// TIA Portal V19 export
FUNCTION "FC_Hilfsfuntionen" : Void   // FC169, LAD
TITLE = Hilfsfunktionen
{ S7_Optimized_Access := 'TRUE' }
// stored: AutoNumber false, SetENOAutomatically true
   VAR_TEMP
      Anf_links : Bool;
      Anf_rechts : Bool;
      Niv_CM01_ok : Bool;
      Niv_CM02_ok : Bool;
      Niv_Spuelen_ok : Bool;
      Fuellstand_ok : Bool;
      Nr : Int;
   END_VAR
   VAR CONSTANT
      Typ_KSoLS : Byte := 16#10;
      Typ_KS : Byte := 16#11;
      Typ_LS : Byte := 16#12;
      Typ_GO_Sperre : Byte := 16#13;
      Typ_GO : Byte := 16#20;
      Ausfahrt : Byte := 16#19;
   END_VAR
BEGIN

REGION Network 1 (SCL): Einfahrsperren / Detailtypen
   REGION CM01
       // CM01 komplett leer
       IF NOT "DB_POS".POS[1].belegt AND NOT NOT "DB_POS".POS[2].belegt AND NOT "DB_POS".POS[3].belegt AND NOT "DB_POS".POS[4].belegt AND NOT "DB_POS".POS[5].belegt AND NOT "DB_POS".POS[6].belegt THEN
           "DB_POS".POS[1].notFG_in := FALSE;
           "DB_POS".POS[2].notFG_in := FALSE;
           "DB_POS".POS[5].notFG_in := FALSE;
           "DB_POS".POS[6].notFG_in := FALSE;
           "DB_POS".POS[1].Detailtyp := #Typ_KSoLS;
           "DB_POS".POS[2].Detailtyp := #Typ_KSoLS;
           "DB_POS".POS[5].Detailtyp := #Typ_KSoLS;
           "DB_POS".POS[6].Detailtyp := #Typ_KSoLS;
       END_IF;
       // Pos.3 (GO) Ziel bzw. belegt
       IF "DB_POS".POS[3].next_WT <> 0 THEN
           "DB_POS".POS[1].notFG_in := TRUE;
           "DB_POS".POS[5].notFG_in := TRUE;
           "DB_POS".POS[1].Detailtyp := #Typ_GO_Sperre;
           "DB_POS".POS[5].Detailtyp := #Typ_GO_Sperre;
       ELSE
           "DB_POS".POS[1].notFG_in := FALSE;
           "DB_POS".POS[5].notFG_in := FALSE;
           "DB_POS".POS[1].Detailtyp := #Typ_KSoLS;
           "DB_POS".POS[5].Detailtyp := #Typ_KSoLS;
       END_IF;
       // Pos.4 (GO) Ziel bzw. belegt 
       IF "DB_POS".POS[4].next_WT <> 0 THEN
           "DB_POS".POS[2].notFG_in := TRUE;
           "DB_POS".POS[6].notFG_in := TRUE;
           "DB_POS".POS[2].Detailtyp := #Typ_GO_Sperre;
           "DB_POS".POS[6].Detailtyp := #Typ_GO_Sperre;
       ELSE
           "DB_POS".POS[2].notFG_in := FALSE;
           "DB_POS".POS[6].notFG_in := FALSE;
           "DB_POS".POS[2].Detailtyp := #Typ_KSoLS;
           "DB_POS".POS[6].Detailtyp := #Typ_KSoLS;
       END_IF;
       //Pos.1/2
       IF ("DB_POS".POS[1].next_WT <> 0) AND ("DB_POS".POS[1].next_WT = "DB_POS".POS[2].next_WT) THEN
           "DB_POS".POS[1].Detailtyp := #Typ_LS;
           "DB_POS".POS[2].Detailtyp := #Typ_LS;
       ELSIF ("DB_POS".POS[1].next_WT <> 0) OR ("DB_POS".POS[2].next_WT <> 0) THEN
           "DB_POS".POS[1].Detailtyp := #Typ_KS;
           "DB_POS".POS[2].Detailtyp := #Typ_KS;
       END_IF;
       //Pos.5/6
       IF ("DB_POS".POS[5].next_WT <> 0) AND ("DB_POS".POS[5].next_WT = "DB_POS".POS[6].next_WT) THEN
           "DB_POS".POS[5].Detailtyp := #Typ_LS;
           "DB_POS".POS[6].Detailtyp := #Typ_LS;
       ELSIF ("DB_POS".POS[5].next_WT <> 0) OR ("DB_POS".POS[6].next_WT <> 0) THEN
           "DB_POS".POS[5].Detailtyp := #Typ_KS;
           "DB_POS".POS[6].Detailtyp := #Typ_KS;
       END_IF;
       //Einfahrsperre Pos.3/4
       "DB_POS".POS[3].notFG_in := ("DB_POS".POS[1].next_WT <> 0) OR ("DB_POS".POS[5].next_WT <> 0);
       "DB_POS".POS[4].notFG_in := ("DB_POS".POS[2].next_WT <> 0) OR ("DB_POS".POS[6].next_WT <> 0);
   END_REGION

   REGION CM03
       // CM03 komplett leer
       IF NOT "DB_POS".POS[7].belegt AND NOT NOT "DB_POS".POS[8].belegt AND NOT "DB_POS".POS[9].belegt AND NOT "DB_POS".POS[10].belegt AND NOT "DB_POS".POS[11].belegt AND NOT "DB_POS".POS[12].belegt THEN
           "DB_POS".POS[7].notFG_in := FALSE;
           "DB_POS".POS[8].notFG_in := FALSE;
           "DB_POS".POS[11].notFG_in := FALSE;
           "DB_POS".POS[12].notFG_in := FALSE;
           "DB_POS".POS[7].Detailtyp := #Typ_KSoLS;
           "DB_POS".POS[8].Detailtyp := #Typ_KSoLS;
           "DB_POS".POS[11].Detailtyp := #Typ_KSoLS;
           "DB_POS".POS[12].Detailtyp := #Typ_KSoLS;
       END_IF;
       // Pos.9 (GO) Ziel bzw. belegt
       IF "DB_POS".POS[9].next_WT <> 0 THEN
           "DB_POS".POS[7].notFG_in := TRUE;
           "DB_POS".POS[11].notFG_in := TRUE;
           "DB_POS".POS[7].Detailtyp := #Typ_GO_Sperre;
           "DB_POS".POS[11].Detailtyp := #Typ_GO_Sperre;
       ELSE
           "DB_POS".POS[7].notFG_in := FALSE;
           "DB_POS".POS[11].notFG_in := FALSE;
           "DB_POS".POS[7].Detailtyp := #Typ_KSoLS;
           "DB_POS".POS[11].Detailtyp := #Typ_KSoLS;
       END_IF;
       // Pos.10 (GO) Ziel bzw. belegt 
       IF "DB_POS".POS[10].next_WT <> 0 THEN
           "DB_POS".POS[8].notFG_in := TRUE;
           "DB_POS".POS[12].notFG_in := TRUE;
           "DB_POS".POS[8].Detailtyp := #Typ_GO_Sperre;
           "DB_POS".POS[12].Detailtyp := #Typ_GO_Sperre;
       ELSE
           "DB_POS".POS[8].notFG_in := FALSE;
           "DB_POS".POS[12].notFG_in := FALSE;
           "DB_POS".POS[8].Detailtyp := #Typ_KSoLS;
           "DB_POS".POS[12].Detailtyp := #Typ_KSoLS;
       END_IF;
       //Pos.7/8
       IF ("DB_POS".POS[7].next_WT <> 0) AND ("DB_POS".POS[7].next_WT = "DB_POS".POS[8].next_WT) THEN
           "DB_POS".POS[7].Detailtyp := #Typ_LS;
           "DB_POS".POS[8].Detailtyp := #Typ_LS;
       ELSIF ("DB_POS".POS[7].next_WT <> 0) OR ("DB_POS".POS[8].next_WT <> 0) THEN
           "DB_POS".POS[7].Detailtyp := #Typ_KS;
           "DB_POS".POS[8].Detailtyp := #Typ_KS;
       END_IF;
       //Pos.11/12
       IF ("DB_POS".POS[11].next_WT <> 0) AND ("DB_POS".POS[11].next_WT = "DB_POS".POS[12].next_WT) THEN
           "DB_POS".POS[11].Detailtyp := #Typ_LS;
           "DB_POS".POS[12].Detailtyp := #Typ_LS;
       ELSIF ("DB_POS".POS[11].next_WT <> 0) OR ("DB_POS".POS[12].next_WT <> 0) THEN
           "DB_POS".POS[11].Detailtyp := #Typ_KS;
           "DB_POS".POS[12].Detailtyp := #Typ_KS;
       END_IF;
       //Einfahrsperre Pos.9/10
       "DB_POS".POS[9].notFG_in := ("DB_POS".POS[7].next_WT <> 0) OR ("DB_POS".POS[11].next_WT <> 0);
       "DB_POS".POS[10].notFG_in := ("DB_POS".POS[8].next_WT <> 0) OR ("DB_POS".POS[12].next_WT <> 0);
   END_REGION

   REGION CM02
       // CM02 komplett leer
       IF NOT "DB_POS".POS[13].belegt AND NOT NOT "DB_POS".POS[14].belegt AND NOT "DB_POS".POS[15].belegt AND NOT "DB_POS".POS[16].belegt AND NOT "DB_POS".POS[17].belegt AND NOT "DB_POS".POS[18].belegt THEN
           "DB_POS".POS[13].notFG_in := FALSE;
           "DB_POS".POS[14].notFG_in := FALSE;
           "DB_POS".POS[17].notFG_in := FALSE;
           "DB_POS".POS[18].notFG_in := FALSE;
           "DB_POS".POS[13].Detailtyp := #Typ_KSoLS;
           "DB_POS".POS[14].Detailtyp := #Typ_KSoLS;
           "DB_POS".POS[17].Detailtyp := #Typ_KSoLS;
           "DB_POS".POS[18].Detailtyp := #Typ_KSoLS;
       END_IF;
       // Pos.15 (GO) Ziel bzw. belegt
       IF "DB_POS".POS[15].next_WT <> 0 THEN
           "DB_POS".POS[13].notFG_in := TRUE;
           "DB_POS".POS[17].notFG_in := TRUE;
           "DB_POS".POS[13].Detailtyp := #Typ_GO_Sperre;
           "DB_POS".POS[17].Detailtyp := #Typ_GO_Sperre;
       ELSE
           "DB_POS".POS[13].notFG_in := FALSE;
           "DB_POS".POS[17].notFG_in := FALSE;
           "DB_POS".POS[13].Detailtyp := #Typ_KSoLS;
           "DB_POS".POS[17].Detailtyp := #Typ_KSoLS;
       END_IF;
       // Pos.16 (GO) Ziel bzw. belegt 
       IF "DB_POS".POS[16].next_WT <> 0 THEN
           "DB_POS".POS[14].notFG_in := TRUE;
           "DB_POS".POS[18].notFG_in := TRUE;
           "DB_POS".POS[14].Detailtyp := #Typ_GO_Sperre;
           "DB_POS".POS[18].Detailtyp := #Typ_GO_Sperre;
       ELSE
           "DB_POS".POS[14].notFG_in := FALSE;
           "DB_POS".POS[18].notFG_in := FALSE;
           "DB_POS".POS[14].Detailtyp := #Typ_KSoLS;
           "DB_POS".POS[18].Detailtyp := #Typ_KSoLS;
       END_IF;
       //Pos.13/14
       IF ("DB_POS".POS[13].next_WT <> 0) AND ("DB_POS".POS[13].next_WT = "DB_POS".POS[14].next_WT) THEN
           "DB_POS".POS[13].Detailtyp := #Typ_LS;
           "DB_POS".POS[14].Detailtyp := #Typ_LS;
       ELSIF ("DB_POS".POS[13].next_WT <> 0) OR ("DB_POS".POS[14].next_WT <> 0) THEN
           "DB_POS".POS[13].Detailtyp := #Typ_KS;
           "DB_POS".POS[14].Detailtyp := #Typ_KS;
       END_IF;
       //Pos.17/18
       IF ("DB_POS".POS[17].next_WT <> 0) AND ("DB_POS".POS[17].next_WT = "DB_POS".POS[18].next_WT) THEN
           "DB_POS".POS[17].Detailtyp := #Typ_LS;
           "DB_POS".POS[18].Detailtyp := #Typ_LS;
       ELSIF ("DB_POS".POS[17].next_WT <> 0) OR ("DB_POS".POS[18].next_WT <> 0) THEN
           "DB_POS".POS[17].Detailtyp := #Typ_KS;
           "DB_POS".POS[18].Detailtyp := #Typ_KS;
       END_IF;
       //Einfahrsperre Pos.15/16
       "DB_POS".POS[15].notFG_in := ("DB_POS".POS[13].next_WT <> 0) OR ("DB_POS".POS[17].next_WT <> 0);
       "DB_POS".POS[16].notFG_in := ("DB_POS".POS[14].next_WT <> 0) OR ("DB_POS".POS[18].next_WT <> 0);
   END_REGION

   REGION CM04
       // CM04 komplett leer
       IF NOT "DB_POS".POS[19].belegt AND NOT NOT "DB_POS".POS[20].belegt AND NOT "DB_POS".POS[21].belegt AND NOT "DB_POS".POS[22].belegt AND NOT "DB_POS".POS[23].belegt AND NOT "DB_POS".POS[24].belegt THEN
           "DB_POS".POS[19].notFG_in := FALSE;
           "DB_POS".POS[20].notFG_in := FALSE;
           "DB_POS".POS[23].notFG_in := FALSE;
           "DB_POS".POS[24].notFG_in := FALSE;
           "DB_POS".POS[19].Detailtyp := #Typ_KSoLS;
           "DB_POS".POS[20].Detailtyp := #Typ_KSoLS;
           "DB_POS".POS[23].Detailtyp := #Typ_KSoLS;
           "DB_POS".POS[24].Detailtyp := #Typ_KSoLS;
       END_IF;
       // Pos.21 (GO) Ziel bzw. belegt
       IF "DB_POS".POS[21].next_WT <> 0 THEN
           "DB_POS".POS[19].notFG_in := TRUE;
           "DB_POS".POS[23].notFG_in := TRUE;
           "DB_POS".POS[19].Detailtyp := #Typ_GO_Sperre;
           "DB_POS".POS[23].Detailtyp := #Typ_GO_Sperre;
       ELSE
           "DB_POS".POS[19].notFG_in := FALSE;
           "DB_POS".POS[23].notFG_in := FALSE;
           "DB_POS".POS[19].Detailtyp := #Typ_KSoLS;
           "DB_POS".POS[23].Detailtyp := #Typ_KSoLS;
       END_IF;
       // Pos.22 (GO) Ziel bzw. belegt 
       IF "DB_POS".POS[22].next_WT <> 0 THEN
           "DB_POS".POS[20].notFG_in := TRUE;
           "DB_POS".POS[24].notFG_in := TRUE;
           "DB_POS".POS[20].Detailtyp := #Typ_GO_Sperre;
           "DB_POS".POS[24].Detailtyp := #Typ_GO_Sperre;
       ELSE
           "DB_POS".POS[20].notFG_in := FALSE;
           "DB_POS".POS[24].notFG_in := FALSE;
           "DB_POS".POS[20].Detailtyp := #Typ_KSoLS;
           "DB_POS".POS[24].Detailtyp := #Typ_KSoLS;
       END_IF;
       //Pos.19/20
       IF ("DB_POS".POS[19].next_WT <> 0) AND ("DB_POS".POS[19].next_WT = "DB_POS".POS[20].next_WT) THEN
           "DB_POS".POS[19].Detailtyp := #Typ_LS;
           "DB_POS".POS[20].Detailtyp := #Typ_LS;
       ELSIF ("DB_POS".POS[19].next_WT <> 0) OR ("DB_POS".POS[20].next_WT <> 0) THEN
           "DB_POS".POS[19].Detailtyp := #Typ_KS;
           "DB_POS".POS[20].Detailtyp := #Typ_KS;
       END_IF;
       //Pos.23/24
       IF ("DB_POS".POS[23].next_WT <> 0) AND ("DB_POS".POS[23].next_WT = "DB_POS".POS[24].next_WT) THEN
           "DB_POS".POS[23].Detailtyp := #Typ_LS;
           "DB_POS".POS[24].Detailtyp := #Typ_LS;
       ELSIF ("DB_POS".POS[23].next_WT <> 0) OR ("DB_POS".POS[24].next_WT <> 0) THEN
           "DB_POS".POS[23].Detailtyp := #Typ_KS;
           "DB_POS".POS[24].Detailtyp := #Typ_KS;
       END_IF;
       //Einfahrsperre Pos.21/22
       "DB_POS".POS[21].notFG_in := ("DB_POS".POS[19].next_WT <> 0) OR ("DB_POS".POS[23].next_WT <> 0);
       "DB_POS".POS[22].notFG_in := ("DB_POS".POS[20].next_WT <> 0) OR ("DB_POS".POS[24].next_WT <> 0);
   END_REGION

   REGION Übergabe
       // Übergabe komplett leer
       IF NOT "DB_POS".POS[25].belegt AND NOT NOT "DB_POS".POS[26].belegt AND NOT "DB_POS".POS[27].belegt AND NOT "DB_POS".POS[28].belegt AND NOT "DB_POS".POS[29].belegt AND NOT "DB_POS".POS[30].belegt THEN
           "DB_POS".POS[25].Detailtyp := #Typ_KSoLS;
           "DB_POS".POS[26].Detailtyp := #Typ_KSoLS;
           "DB_POS".POS[29].Detailtyp := #Typ_KSoLS;
           "DB_POS".POS[30].Detailtyp := #Typ_KSoLS;
       END_IF;
       // Pos.27 (GO) Ziel bzw. belegt
       IF "DB_POS".POS[27].next_WT <> 0 THEN
           "DB_POS".POS[25].Detailtyp := #Typ_GO_Sperre;
           "DB_POS".POS[29].Detailtyp := #Typ_GO_Sperre;
       ELSE
           "DB_POS".POS[25].Detailtyp := #Typ_KSoLS;
           "DB_POS".POS[29].Detailtyp := #Typ_KSoLS;
       END_IF;
       // Pos.22 (GO) Ziel bzw. belegt 
       IF "DB_POS".POS[28].next_WT <> 0 THEN
           "DB_POS".POS[26].Detailtyp := #Typ_GO_Sperre;
           "DB_POS".POS[30].Detailtyp := #Typ_GO_Sperre;
       ELSE
           "DB_POS".POS[26].Detailtyp := #Typ_KSoLS;
           "DB_POS".POS[30].Detailtyp := #Typ_KSoLS;
       END_IF;
       //Pos.25/26
       IF ("DB_POS".POS[25].next_WT <> 0) AND ("DB_POS".POS[25].next_WT = "DB_POS".POS[26].next_WT) THEN
           "DB_POS".POS[25].Detailtyp := #Typ_LS;
           "DB_POS".POS[26].Detailtyp := #Typ_LS;
       ELSIF ("DB_POS".POS[25].next_WT <> 0) OR ("DB_POS".POS[26].next_WT <> 0) THEN
           "DB_POS".POS[25].Detailtyp := #Typ_KS;
           "DB_POS".POS[26].Detailtyp := #Typ_KS;
       END_IF;
       //Pos.29/30
       IF ("DB_POS".POS[29].next_WT <> 0) AND ("DB_POS".POS[29].next_WT = "DB_POS".POS[30].next_WT) THEN
           "DB_POS".POS[29].Detailtyp := #Typ_LS;
           "DB_POS".POS[30].Detailtyp := #Typ_LS;
       ELSIF ("DB_POS".POS[29].next_WT <> 0) OR ("DB_POS".POS[30].next_WT <> 0) THEN
           "DB_POS".POS[29].Detailtyp := #Typ_KS;
           "DB_POS".POS[30].Detailtyp := #Typ_KS;
       END_IF;

   END_REGION
END_REGION

REGION Network 2 (SCL): Deckelanforderungen

   REGION CM01
       #Anf_links := FALSE;
       #Anf_rechts := FALSE;

       // Check Quelle
       IF ("DB_POS".POS[1].Quelle AND ("DB_POS".POS[1].WT_DB <> 0)) OR
          ("DB_POS".POS[3].Quelle AND ("DB_POS".POS[3].WT_DB <> 0)) OR
          ("DB_POS".POS[5].Quelle AND  ("DB_POS".POS[5].WT_DB <> 0)) THEN
           #Anf_links := TRUE;
       END_IF;

       IF ("DB_POS".POS[2].Quelle AND ("DB_POS".POS[2].WT_DB <> 0)) OR
           ("DB_POS".POS[4].Quelle AND ("DB_POS".POS[4].WT_DB <> 0)) OR
           ("DB_POS".POS[6].Quelle AND  ("DB_POS".POS[6].WT_DB <> 0)) THEN
           #Anf_rechts := TRUE;
       END_IF;

       IF "DB_POS".POS[1].Quelle AND ("DB_POS".POS[1].WT_DB <> 0) AND ("DB_POS".POS[1].WT_DB = "DB_POS".POS[2].WT_DB) THEN
           #Anf_rechts := TRUE;
       END_IF;

       IF "DB_POS".POS[5].Quelle AND ("DB_POS".POS[5].WT_DB <> 0) AND ("DB_POS".POS[5].WT_DB = "DB_POS".POS[6].WT_DB) THEN
           #Anf_rechts := TRUE;
       END_IF;

       // Check Ziel
       IF (("DB_POS".POS[1].Ziel AND ("DB_POS".POS[1].next_WT <> 0)) OR ("DB_POS".POS[3].Ziel AND ("DB_POS".POS[3].next_WT <> 0)) OR ("DB_POS".POS[5].Ziel AND  ("DB_POS".POS[5].next_WT <> 0))) AND "DI_FW_1".ZST.Oben_li THEN
           #Anf_links := TRUE;
       END_IF;

       IF (("DB_POS".POS[2].Ziel AND ("DB_POS".POS[2].next_WT <> 0)) OR ("DB_POS".POS[4].Ziel AND ("DB_POS".POS[4].next_WT <> 0)) OR ("DB_POS".POS[6].Ziel AND  ("DB_POS".POS[6].next_WT <> 0)))  AND "DI_FW_1".ZST.Oben_re THEN
           #Anf_rechts := TRUE;
       END_IF;

       IF "DB_POS".POS[1].Ziel AND ("DB_POS".POS[1].next_WT <> 0) AND ("DB_POS".POS[1].next_WT = "DB_POS".POS[2].next_WT)  AND "DI_FW_1".ZST.Oben_re THEN
           #Anf_rechts := TRUE;
       END_IF;

       IF "DB_POS".POS[5].Ziel AND ("DB_POS".POS[5].next_WT <> 0) AND ("DB_POS".POS[5].next_WT = "DB_POS".POS[6].next_WT)  AND "DI_FW_1".ZST.Oben_re THEN
           #Anf_rechts := TRUE;
       END_IF;
       //
       IF #Anf_links THEN
           "Deckel_CM01".Zst.Req_links_auf := TRUE;
       ELSIF "Deckel_CM01".Zst.TW_sicher THEN
           "Deckel_CM01".Zst.Req_links_auf := FALSE;
       END_IF;

       IF #Anf_rechts THEN
           "Deckel_CM01".Zst.Req_rechts_auf := TRUE;
       ELSIF "Deckel_CM01".Zst.TW_sicher THEN
           "Deckel_CM01".Zst.Req_rechts_auf := FALSE;
       END_IF;

   END_REGION

   REGION CM02
       #Anf_links := FALSE;
       #Anf_rechts := FALSE;

       // Check Quelle
       IF ("DB_POS".POS[13].Quelle AND ("DB_POS".POS[13].WT_DB <> 0)) OR
           ("DB_POS".POS[15].Quelle AND ("DB_POS".POS[15].WT_DB <> 0)) OR
           ("DB_POS".POS[17].Quelle AND  ("DB_POS".POS[17].WT_DB <> 0)) THEN
           #Anf_links := TRUE;
       END_IF;

       IF ("DB_POS".POS[14].Quelle AND ("DB_POS".POS[14].WT_DB <> 0)) OR
           ("DB_POS".POS[16].Quelle AND ("DB_POS".POS[16].WT_DB <> 0)) OR
           ("DB_POS".POS[18].Quelle AND ("DB_POS".POS[18].WT_DB <> 0)) THEN
           #Anf_rechts := TRUE;
       END_IF;

       IF "DB_POS".POS[13].Quelle AND ("DB_POS".POS[13].WT_DB <> 0) AND ("DB_POS".POS[13].WT_DB = "DB_POS".POS[14].WT_DB) THEN
           #Anf_rechts := TRUE;
       END_IF;

       IF "DB_POS".POS[17].Quelle AND ("DB_POS".POS[17].WT_DB <> 0) AND ("DB_POS".POS[17].WT_DB = "DB_POS".POS[18].WT_DB) THEN
           #Anf_rechts := TRUE;
       END_IF;

       // Check Ziel
       IF (("DB_POS".POS[13].Ziel AND ("DB_POS".POS[13].next_WT <> 0)) OR ("DB_POS".POS[15].Ziel AND ("DB_POS".POS[15].next_WT <> 0)) OR ("DB_POS".POS[17].Ziel AND  ("DB_POS".POS[17].next_WT <> 0))) AND "DI_FW_1".ZST.Oben_li THEN
           #Anf_links := TRUE;
       END_IF;

       IF (("DB_POS".POS[14].Ziel AND ("DB_POS".POS[14].next_WT <> 0)) OR ("DB_POS".POS[16].Ziel AND ("DB_POS".POS[16].next_WT <> 0)) OR ("DB_POS".POS[18].Ziel AND  ("DB_POS".POS[18].next_WT <> 0))) AND "DI_FW_1".ZST.Oben_re THEN
           #Anf_rechts := TRUE;
       END_IF;

       IF "DB_POS".POS[13].Ziel  AND ("DB_POS".POS[13].next_WT <> 0) AND ("DB_POS".POS[13].next_WT = "DB_POS".POS[14].next_WT) AND "DI_FW_1".ZST.Oben_re THEN
           #Anf_rechts := TRUE;
       END_IF;

       IF "DB_POS".POS[17].Ziel AND ("DB_POS".POS[17].next_WT <> 0) AND ("DB_POS".POS[17].next_WT = "DB_POS".POS[18].next_WT) AND "DI_FW_1".ZST.Oben_re THEN
           #Anf_rechts := TRUE;
       END_IF;
       //
       IF #Anf_links THEN
           "Deckel_CM02".Zst.Req_links_auf := TRUE;
       ELSIF "Deckel_CM02".Zst.TW_sicher THEN
           "Deckel_CM02".Zst.Req_links_auf := FALSE;
       END_IF;

       IF #Anf_rechts THEN
           "Deckel_CM02".Zst.Req_rechts_auf := TRUE;
       ELSIF "Deckel_CM02".Zst.TW_sicher THEN
           "Deckel_CM02".Zst.Req_rechts_auf := FALSE;
       END_IF;

   END_REGION
END_REGION

REGION Network 3 (SCL): Anforderung Rolltor
   "Tor".Zst.Req_Auf := ("DI_QF_WR02_03".Zst.Req_WR02_In
   OR "DI_QF_WR02_03".Zst.Req_WR03_In
   OR "DI_QF_WR02_03".Zst.Req_WR02_Out
   OR "DI_QF_WR02_03".Zst.Req_WR03_Out) AND "DI_QF_WR02_03".Zst.TW_sicher;
END_REGION

REGION Network 4 (SCL): Keine Einfahrt / kein neuer Befehl / Freigabe Ausfahrt

   // Freigabe Abluft, kein Notstrom, kein Gasalarm
   "DI_FW_Auftrag_DB".Frg_Ablauf := "DB_PNOZ_IN_Out".In.Abluft_ok AND "E_Frg_AbLW" AND "E_DL_min_ok" AND "E_Al_Gas_ok" AND NOT "E_Not-Strom" AND "E_Normal-Vers";

   //Füllstand der Becken ok, erst dann Einfahren 
   //Beide Spülbecken + 1 Säurebecken muss Niveau haben --> Signale Niveau_ok Verzögert + entsprechende Meldung
   #Niv_CM01_ok := NOT "DB_NSP".NSP[1].AM_AL_min AND "E_Niv_UeL_CM01.BL01";
   #Niv_CM02_ok := NOT "DB_NSP".NSP[13].AM_AL_min  AND  "E_Niv_UeL_CM02.BL08";
   #Niv_Spuelen_ok := NOT "DB_NSP".NSP[19].AM_AL_min;
   #Fuellstand_ok := (#Niv_CM01_ok OR #Niv_CM02_ok) AND #Niv_Spuelen_ok;

   // Kein eingeschränkter Betrieb Abluftwäscher VEW-Waser und Füllstand
   "DI_FW_Auftrag_DB".Frg_Einfahrt := "E_kein_NB_AblW" AND "DI_FW_Auftrag_DB".Frg_Ablauf AND #Fuellstand_ok AND "E_VEW_ok";

   // Freigabe Fertig-Korb 
   IF (("DB_WT1".akt_CMD = #Ausfahrt AND "DB_POS".POS["DB_WT1".POS].fertig) OR ("DB_WT2".akt_CMD = #Ausfahrt AND "DB_POS".POS["DB_WT2".POS].fertig) OR
       ("DB_WT3".akt_CMD = #Ausfahrt AND "DB_POS".POS["DB_WT3".POS].fertig) OR ("DB_WT4".akt_CMD = #Ausfahrt AND "DB_POS".POS["DB_WT4".POS].fertig) OR
       ("DB_WT5".akt_CMD = #Ausfahrt AND "DB_POS".POS["DB_WT5".POS].fertig) OR ("DB_WT6".akt_CMD = #Ausfahrt AND "DB_POS".POS["DB_WT6".POS].fertig) OR
       ("DB_WT7".akt_CMD = #Ausfahrt AND "DB_POS".POS["DB_WT7".POS].fertig) OR ("DB_WT8".akt_CMD = #Ausfahrt AND "DB_POS".POS["DB_WT8".POS].fertig) OR
       ("DB_WT9".akt_CMD = #Ausfahrt AND "DB_POS".POS["DB_WT9".POS].fertig) OR ("DB_WT10".akt_CMD = #Ausfahrt AND "DB_POS".POS["DB_WT10".POS].fertig) OR
       ("DB_WT11".akt_CMD = #Ausfahrt AND "DB_POS".POS["DB_WT11".POS].fertig) OR ("DB_WT12".akt_CMD = #Ausfahrt AND "DB_POS".POS["DB_WT12".POS].fertig))
       AND "E_T_Frg_BE"  AND "E_VEW_ok" AND "E_DL_min_ok" THEN
       "DI_FW_Auftrag_DB".Frg_Ausfahrt := TRUE;
   END_IF;
END_REGION

REGION Network 5 (SCL): Einfahsprerren CM01 / CM02
   // CM01
   "DB_POS".POS[1].Sperre_in := "Panel".CM01.Wartung;
   "DB_POS".POS[2].Sperre_in := "Panel".CM01.Wartung;
   "DB_POS".POS[3].Sperre_in := "Panel".CM01.Wartung;
   "DB_POS".POS[4].Sperre_in := "Panel".CM01.Wartung;
   "DB_POS".POS[5].Sperre_in := "Panel".CM01.Wartung;
   "DB_POS".POS[6].Sperre_in := "Panel".CM01.Wartung;

   // Übervoll (Sperre setzend - siehe NW1)
   IF NOT "E_Niv_UeL_CM01.BL01" THEN
       "DB_POS".POS[1].notFG_in := TRUE;
       "DB_POS".POS[2].notFG_in := TRUE;
       "DB_POS".POS[3].notFG_in := TRUE;
       "DB_POS".POS[4].notFG_in := TRUE;
       "DB_POS".POS[5].notFG_in := TRUE;
       "DB_POS".POS[6].notFG_in := TRUE;
   END_IF;

   // CM02
   "DB_POS".POS[13].Sperre_in := "Panel".CM02.Wartung;
   "DB_POS".POS[14].Sperre_in := "Panel".CM02.Wartung;
   "DB_POS".POS[15].Sperre_in := "Panel".CM02.Wartung;
   "DB_POS".POS[16].Sperre_in := "Panel".CM02.Wartung;
   "DB_POS".POS[17].Sperre_in := "Panel".CM02.Wartung;
   "DB_POS".POS[18].Sperre_in := "Panel".CM02.Wartung;

   // Übervoll (Sperre setzend - siehe NW1)
   IF NOT "E_Niv_UeL_CM02.BL08" THEN
       "DB_POS".POS[13].notFG_in := TRUE;
       "DB_POS".POS[14].notFG_in := TRUE;
       "DB_POS".POS[15].notFG_in := TRUE;
       "DB_POS".POS[16].notFG_in := TRUE;
       "DB_POS".POS[17].notFG_in := TRUE;
       "DB_POS".POS[18].notFG_in := TRUE;
   END_IF;
END_REGION

REGION Network 6 (SCL): Sperren Kombibetrieb GO CM02 / CM04
   IF NOT "DB_ANLAGE".config.NormalB THEN
       // CM02
       "DB_POS".POS[15].Sperre_in := TRUE;
       "DB_POS".POS[16].Sperre_in := TRUE;
       // CM04
       "DB_POS".POS[21].Sperre_in := TRUE;
       "DB_POS".POS[22].Sperre_in := TRUE;
   END_IF;
END_REGION

REGION Network 7 (SCL): Positionsincremente
   // Ungerade --> gerade

   "DB_POS".POS[2].IncPos := "DB_POS".POS[1].IncPos;
   "DB_POS".POS[4].IncPos := "DB_POS".POS[3].IncPos;
   "DB_POS".POS[6].IncPos := "DB_POS".POS[5].IncPos;
   "DB_POS".POS[8].IncPos := "DB_POS".POS[7].IncPos;
   "DB_POS".POS[10].IncPos := "DB_POS".POS[9].IncPos;
   "DB_POS".POS[12].IncPos := "DB_POS".POS[11].IncPos;
   "DB_POS".POS[14].IncPos := "DB_POS".POS[13].IncPos;
   "DB_POS".POS[16].IncPos := "DB_POS".POS[15].IncPos;
   "DB_POS".POS[18].IncPos := "DB_POS".POS[17].IncPos;
   "DB_POS".POS[20].IncPos := "DB_POS".POS[19].IncPos;
   "DB_POS".POS[22].IncPos := "DB_POS".POS[21].IncPos;
   "DB_POS".POS[24].IncPos := "DB_POS".POS[23].IncPos;
   "DB_POS".POS[26].IncPos := "DB_POS".POS[25].IncPos;
   "DB_POS".POS[28].IncPos := "DB_POS".POS[27].IncPos;
   "DB_POS".POS[30].IncPos := "DB_POS".POS[29].IncPos;
END_REGION

REGION Network 8 (SCL): Korbumläufe Meldungen
   FOR #Nr := "KorbAnzahl_min" TO "KorbAnzahl_max" DO
       IF "DB_Korbumlaeufe".Korb[#Nr].Durchlaeufe >= "DB_Korbumlaeufe".Korb[#Nr].max_Durchlaeufe THEN
           "DB_Korbumlaeufe".Korb[#Nr].max_erreicht := TRUE;
           "DB_Korbumlaeufe".Korb[#Nr].Warnung := FALSE;
       ELSIF ("DB_Korbumlaeufe".Korb[#Nr].Durchlaeufe >= ("DB_Korbumlaeufe".Korb[#Nr].max_Durchlaeufe - 3)) AND NOT "DB_Korbumlaeufe".Korb[#Nr].max_erreicht THEN
           "DB_Korbumlaeufe".Korb[#Nr].Warnung := TRUE;
       ELSE
           "DB_Korbumlaeufe".Korb[#Nr].max_erreicht := FALSE;
           "DB_Korbumlaeufe".Korb[#Nr].Warnung := FALSE;
       END_IF;
   END_FOR;
END_REGION

REGION Network 9 (SCL): Bits für Anzeige Materialcheck
   // Modus auswerten
   IF NOT "DB_ANLAGE".config.NormalB THEN
       // Kombi-Mode
       CASE "DB_Prog_edit".Prog_Aufgabe.Korb_Nr OF
           1..3:  // "151" Korb kurz 1..3
               "Panel".Betriebsmodus.Korb_151 := TRUE;
               "Panel".Betriebsmodus.Korb_161 := FALSE;

           4..8:   // "161" Korb kurz 4..8
               "Panel".Betriebsmodus.Korb_151 := FALSE;
               "Panel".Betriebsmodus.Korb_161 := TRUE;

           9..11:  // "151" Korb lang 1..3
               "Panel".Betriebsmodus.Korb_151 := TRUE;
               "Panel".Betriebsmodus.Korb_161 := FALSE;

           12..13:   // "161" Korb lang 4, Großoptik 
               "Panel".Betriebsmodus.Korb_151 := FALSE;
               "Panel".Betriebsmodus.Korb_161 := TRUE;
       END_CASE;

   ELSE
       // Normalbetrieb
       "Panel".Betriebsmodus.Korb_151 := FALSE;
       "Panel".Betriebsmodus.Korb_161 := FALSE;
   END_IF;
END_REGION
END_FUNCTION
